// SIMATIC S7-200 SMART project (STEP 7-Micro/WIN SMART), CPU SR40

SYMBOL_TABLE 系统符号
Always_On        SM0.0    // 始终接通
Last_Scan        SMW22    // 最后一次扫描循环的扫描时间
END_SYMBOL_TABLE

SUBROUTINE_BLOCK Time_Clock1:SBR0
TITLE=子程序注释
VAR_INPUT
Stare:BOOL;	// L0.0 定时器启动信号
Stare_Pulse:BOOL;	// L0.1 该定时器输入脉冲信号，只能使用SM0.5 一秒的脉冲边沿信号作为时基
Set_Time:WORD;	// LW1 设定时间，时基为1秒
END_VAR
VAR_IN_OUT
Now_Time:WORD;	// LW3 当前时间
END_VAR
VAR_OUTPUT
Result:BOOL;	// L5.0 定时器定时完成信号
END_VAR
BEGIN
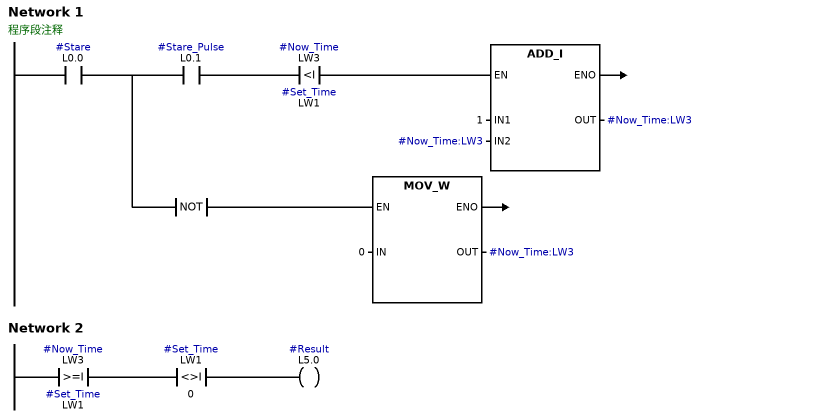
Network 1
// 程序段注释
LD     #Stare:L0.0
LPS
A      #Stare_Pulse:L0.1
AW<    #Now_Time:LW3, #Set_Time:LW1
+I     1, #Now_Time:LW3
LPP
NOT
MOVW   0, #Now_Time:LW3
Network 2
LDW>=  #Now_Time:LW3, #Set_Time:LW1
AW<>   #Set_Time:LW1, 0
=      #Result:L5.0
END_SUBROUTINE_BLOCK

SUBROUTINE_BLOCK 指针:SBR1
TITLE=子程序注释
BEGIN
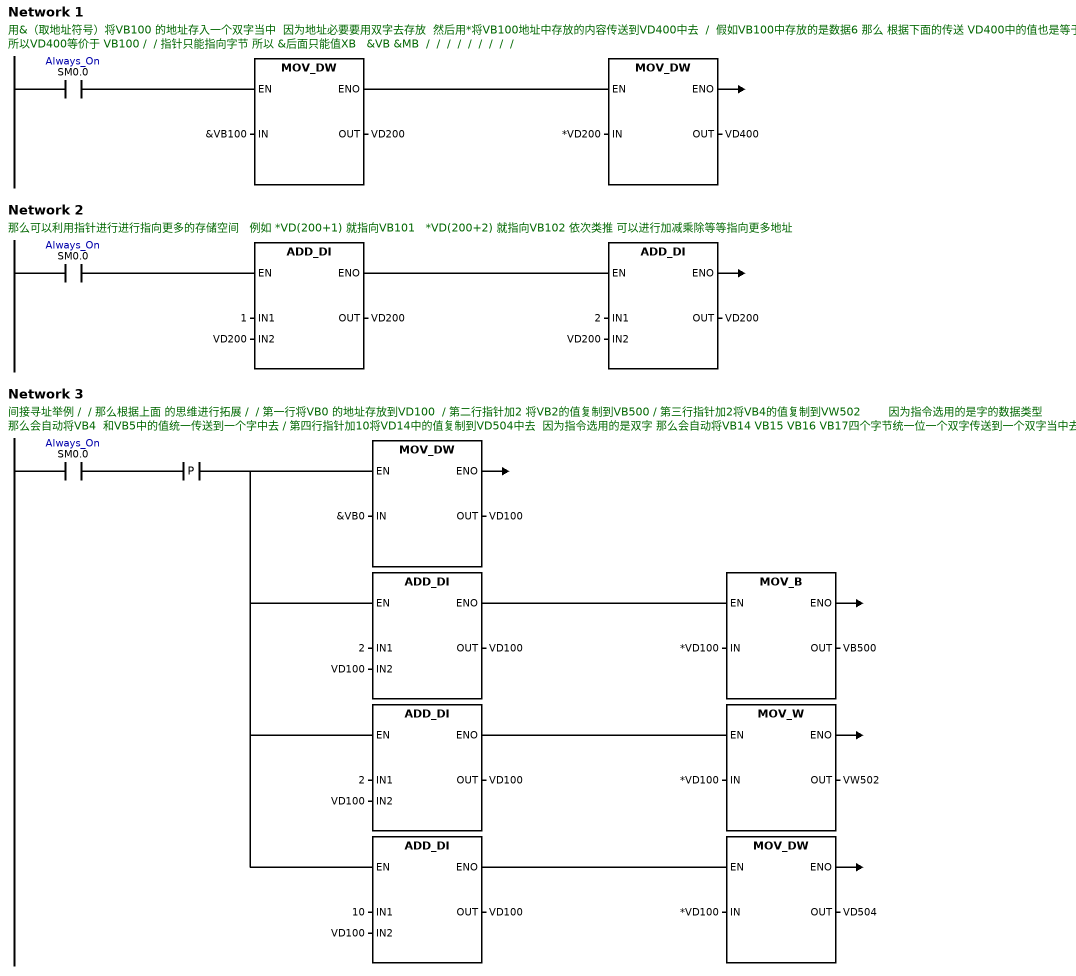
Network 1
// 用&（取地址符号）将VB100 的地址存入一个双字当中  因为地址必要要用双字去存放  然后用*将VB100地址中存放的内容传送到VD400中去 
//  假如VB100中存放的是数据6 那么 根据下面的传送 VD400中的值也是等于6  所以VD400等价于 VB100
// 
// 指针只能指向字节 所以 &后面只能值XB   &VB &MB 
// 
// 
// 
// 
// 
// 
// 
// 
// 
LD     Always_On:SM0.0
MOVD   &VB100, VD200
AENO
MOVD   *VD200, VD400
Network 2
// 那么可以利用指针进行进行指向更多的存储空间   例如 *VD(200+1) 就指向VB101   *VD(200+2) 就指向VB102 依次类推 可以进行加减乘除等等指向更多地址
LD     Always_On:SM0.0
+D     1, VD200
AENO
+D     2, VD200
Network 3
// 间接寻址举例
// 
// 那么根据上面 的思维进行拓展
// 
// 第一行将VB0 的地址存放到VD100 
// 第二行指针加2 将VB2的值复制到VB500
// 第三行指针加2将VB4的值复制到VW502        因为指令选用的是字的数据类型 那么会自动将VB4  和VB5中的值统一传送到一个字中去
// 第四行指针加10将VD14中的值复制到VD504中去  因为指令选用的是双字 那么会自动将VB14 VB15 VB16 VB17四个字节统一位一个双字传送到一个双字当中去
// 
// 
//    
// (network saved uncompiled; LAD cells follow)
// row 0: c0 -| |- Always_On:SM0.0  c1 -|P|-  v  c2 --  c3 [MOV_DW EN:=power@row0, IN:=&VB0, ENO=>power, OUT=>VD100]  c4 ->
// row 1: c1 ^v  c3 [box]
// row 2: c1 ^v  c2 --  c3 [ADD_DI EN:=power@row2, IN1:=2, IN2:=VD100, ENO=>power, OUT=>VD100]  c4 --  c5 --  c6 [MOV_B EN:=power@row2, IN:=*VD100, ENO=>power, OUT=>VB500]  c7 ->
// row 3: c1 ^v  c3 [box]  c6 [box]
// row 4: c1 ^v  c2 --  c3 [ADD_DI EN:=power@row4, IN1:=2, IN2:=VD100, ENO=>power, OUT=>VD100]  c4 --  c5 --  c6 [MOV_W EN:=power@row4, IN:=*VD100, ENO=>power, OUT=>VW502]  c7 ->
// row 5: c1 ^v  c3 [box]  c6 [box]
// row 6: c1 ^  c2 --  c3 [ADD_DI EN:=power@row6, IN1:=10, IN2:=VD100, ENO=>power, OUT=>VD100]  c4 --  c5 --  c6 [MOV_DW EN:=power@row6, IN:=*VD100, ENO=>power, OUT=>VD504]  c7 ->
// row 7: c3 [box]  c6 [box]
END_SUBROUTINE_BLOCK

SUBROUTINE_BLOCK Time_Clock2:SBR2
TITLE=该计时方法受扫描周期的影响，所以回存在几百毫秒的误差 单字
VAR_INPUT
Star:BOOL;	// L0.0 计时启动信号
Set_Time:WORD;	// LW1 设定时间
END_VAR
VAR_IN_OUT
Now_Time:WORD;	// LW3 当前时间
END_VAR
VAR_OUTPUT
Result:BOOL;	// L5.0 定时完成，定时器输出结果
END_VAR
BEGIN
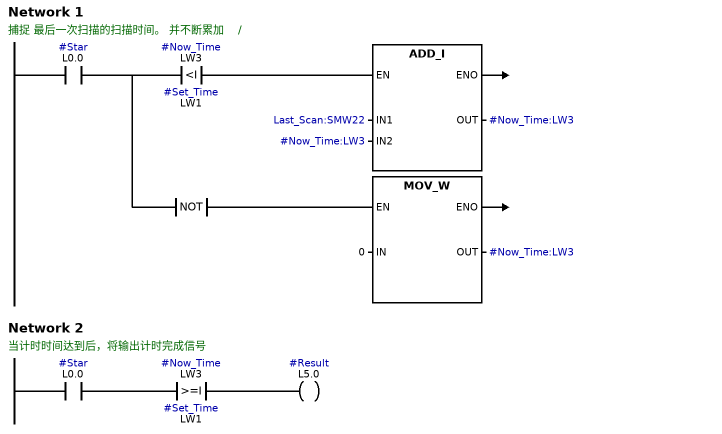
Network 1
// 捕捉 最后一次扫描的扫描时间。 并不断累加   
// 
LD     #Star:L0.0
LPS
AW<    #Now_Time:LW3, #Set_Time:LW1
+I     Last_Scan:SMW22, #Now_Time:LW3
LPP
NOT
MOVW   0, #Now_Time:LW3
Network 2
// 当计时时间达到后，将输出计时完成信号
LD     #Star:L0.0
AW>=   #Now_Time:LW3, #Set_Time:LW1
=      #Result:L5.0
END_SUBROUTINE_BLOCK

SUBROUTINE_BLOCK Time_Clock3:SBR3
TITLE=
VAR_INPUT
Star:BOOL;	// L0.0 计算间隔时间指令计算当前时间与 IN 中提供的时间的时间差，然后将差值存储在 OUT 中
Star_Pulse:BOOL;	// L0.1 开始间隔时间指令读取内置 1 毫秒计数器的当前值，并将该值存储在 OUT 中。 双字毫秒
Set_Time:DWORD;	// LD1 设定时间
END_VAR
VAR_IN_OUT
Now_Time:DWORD;	// LD5 时间差
END_VAR
VAR_OUTPUT
Result:BOOL;	// L9.0 定时器定时完成输出信号
END_VAR
VAR
Star_Time:DWORD;	// LD10 开始时间
END_VAR
BEGIN
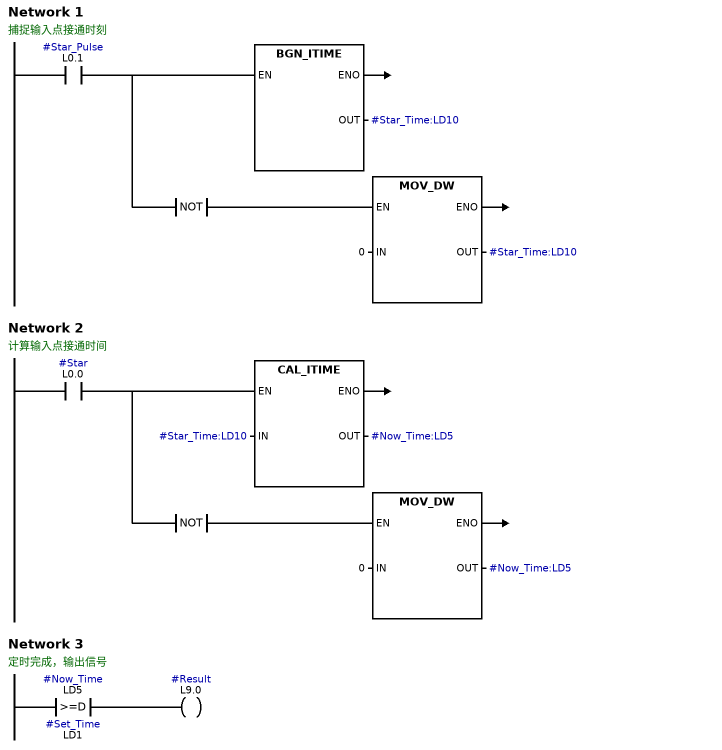
Network 1
// 捕捉输入点接通时刻
LD     #Star_Pulse:L0.1
BITIM  #Star_Time:LD10
NOT
MOVD   0, #Star_Time:LD10
Network 2
// 计算输入点接通时间
LD     #Star:L0.0
CITIM  #Star_Time:LD10, #Now_Time:LD5
NOT
MOVD   0, #Now_Time:LD5
Network 3
// 定时完成，输出信号
LDD>=  #Now_Time:LD5, #Set_Time:LD1
=      #Result:L9.0
END_SUBROUTINE_BLOCK
